FUNCTION_BLOCK FB_MotorContactor 
VAR
	Output AT %Q* : BOOL;
END_VAR

METHOD SwitchOff : BOOL
VAR_INPUT
END_VAR
Output := FALSE;
END_METHOD

METHOD SwitchOn : BOOL
VAR_INPUT
END_VAR
Output := TRUE;
END_METHOD

END_FUNCTION_BLOCK

(* stored: Version 1.1.0.1, ProductVersion 3.1.4024.9
   POU FB_MotorContactor: Id {43b85ac7-8b1f-46e0-bcc2-7590801b4a39}, SpecialFunc None
   Method SwitchOff: Id {d29289eb-8511-4575-8523-c2a0ccb2babf}
   Method SwitchOn: Id {9a2dafc0-873a-49ec-92ef-38112ab95995} *)
